(* PLC project MotionTest1, Higen MCL 1 *)
(* stored: creationDateTime 2012-01-06T15:20:13, modificationDateTime 2013-05-16T00:05:34 *)

FUNCTION_BLOCK wxgetval
  VAR
    getpy : python_gear;
    latch : SR;
  END_VAR
  VAR_INPUT
    name : STRING;
  END_VAR
  VAR_OUTPUT
    val : BOOL;
  END_VAR
  VAR  (* added by the conversion: wires and edge detectors of the diagram *)
    _EQ41_ENO : BOOL;
    _EQ41_OUT : BOOL;
    _EQ3_ENO : BOOL;
    _EQ3_OUT : BOOL;
  END_VAR

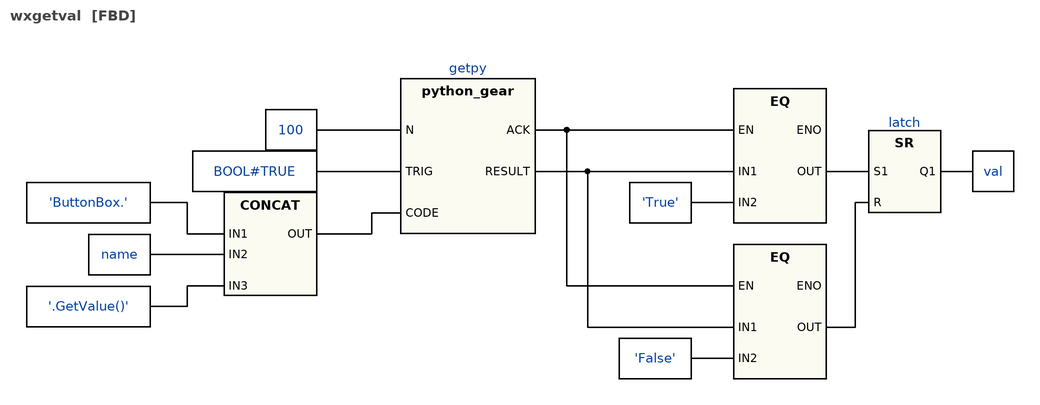
(* FBD diagram, written out as Structured Text *)
getpy(N := 100, TRIG := BOOL#TRUE, CODE := CONCAT('ButtonBox.', name, '.GetValue()'));
_EQ41_OUT := EQ(EN := getpy.ACK, IN1 := getpy.RESULT, IN2 := 'True', ENO => _EQ41_ENO);
_EQ3_OUT := EQ(EN := getpy.ACK, IN1 := getpy.RESULT, IN2 := 'False', ENO => _EQ3_ENO);
latch(S1 := _EQ41_OUT, R := _EQ3_OUT);
val := latch.Q1;
END_FUNCTION_BLOCK

(* -- *)
PROGRAM main
  VAR
    Done : BOOL;
    Slave : AXIS_REF;
    Master1 : AXIS_REF;
    Master2 : AXIS_REF;
    switch : MC_Power;
    readpos : MC_ReadActualPosition;
    sPn : LREAL;
    m1Pn : LREAL;
    m2Pn : LREAL;
    sVn : LREAL;
    m1Vn : LREAL;
    m2Vn : LREAL;
    setpos : MC_SetPosition;
    readspeed : MC_ReadParameter;
    sim : MC_Sim;
    bt1 : wxgetval;
    Block1 : wxgetval;
    Block2 : wxgetval;
    Block3 : wxgetval;
    Block6 : wxgetval;
    MC_Sim0 : MC_Sim;
    MC_Power0 : MC_Power;
    MC_ReadActualPosition0 : MC_ReadActualPosition;
    MC_SetPosition0 : MC_SetPosition;
    MC_ReadParameter0 : MC_ReadParameter;
    MC_MoveAbsolute0 : MC_MoveAbsolute;
    MC_Sim1 : MC_Sim;
    MC_ReadActualPosition1 : MC_ReadActualPosition;
    MC_ReadParameter1 : MC_ReadParameter;
    MC_Power1 : MC_Power;
    MC_SetPosition1 : MC_SetPosition;
    MC_MoveAbsolute1 : MC_MoveAbsolute;
    MC_MoveAbsolute2 : MC_MoveAbsolute;
    MC_MoveAbsolute3 : MC_MoveAbsolute;
    MC_MoveAbsolute4 : MC_MoveAbsolute;
    MC_MoveAbsolute5 : MC_MoveAbsolute;
    MC_CombineAxes0 : MC_CombineAxes;
    MC_Stop0 : MC_Stop;
    MC_Stop1 : MC_Stop;
    MC_Stop2 : MC_Stop;
  END_VAR

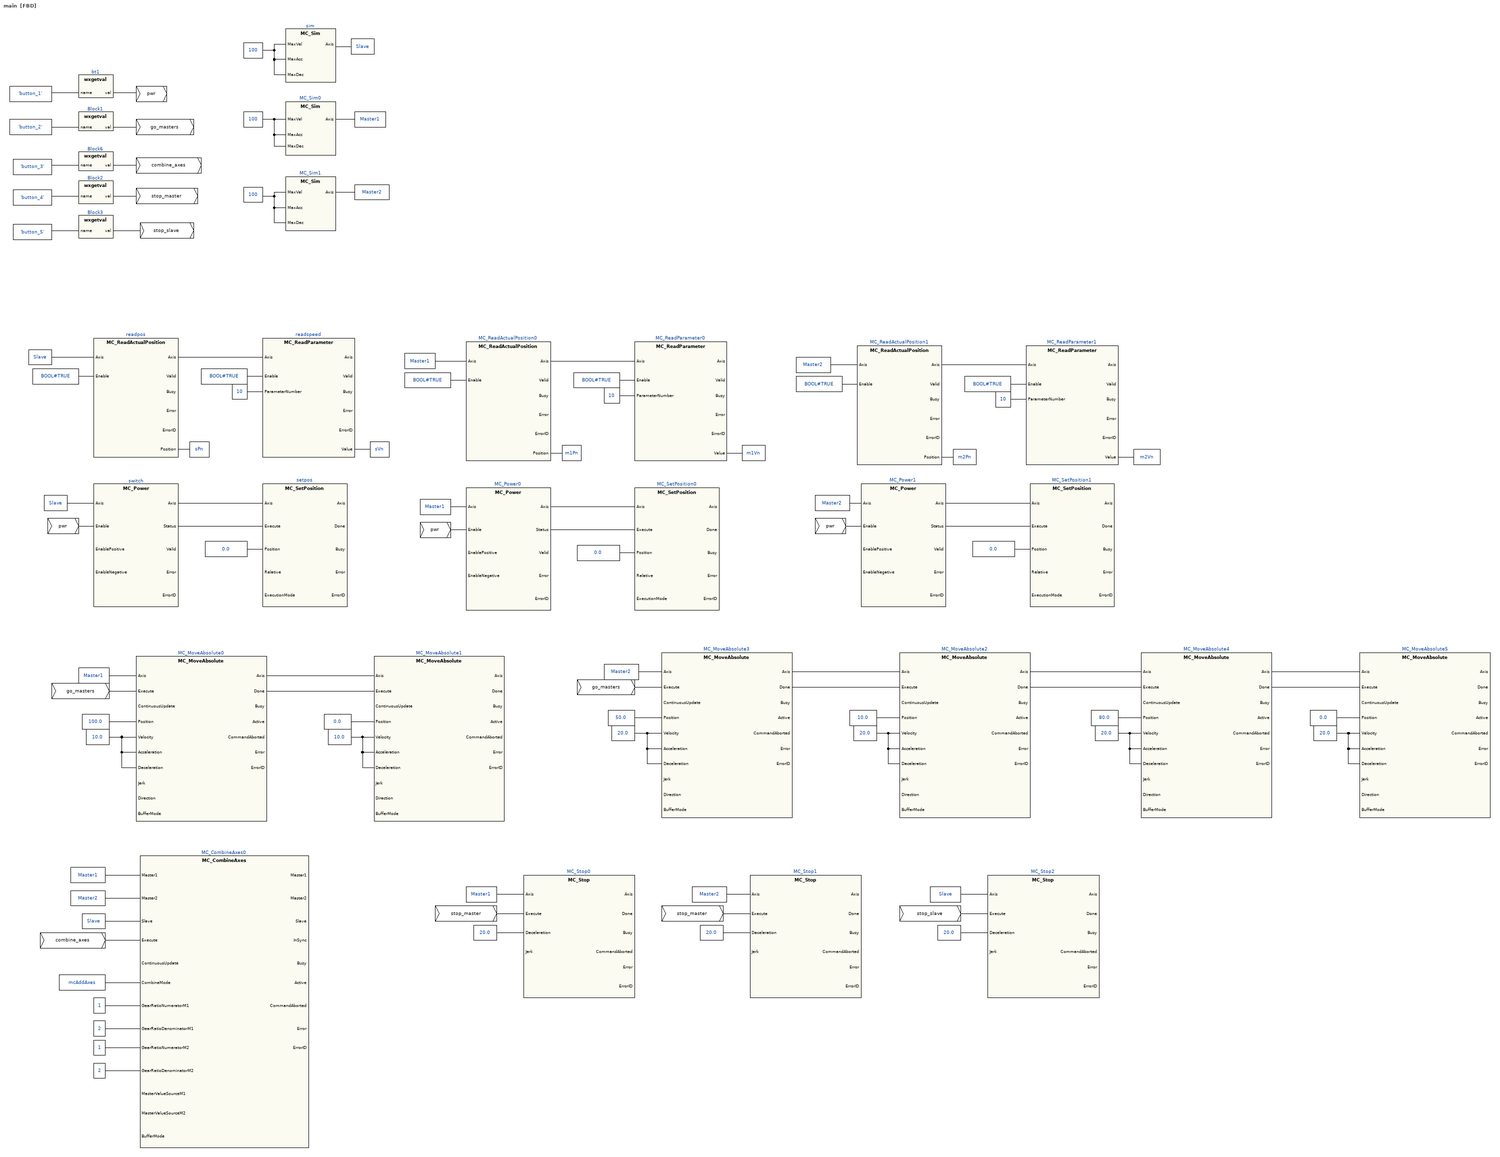
(* FBD diagram, written out as Structured Text *)
sim(MaxVel := 100, MaxAcc := 100, MaxDec := 100);
Slave := sim.Axis;
MC_Sim0(MaxVel := 100, MaxAcc := 100, MaxDec := 100);
Master1 := MC_Sim0.Axis;
MC_Sim1(MaxVel := 100, MaxAcc := 100, MaxDec := 100);
Master2 := MC_Sim1.Axis;
readpos(Axis := Slave, Enable := BOOL#TRUE);
sPn := readpos.Position;
readspeed(Axis := readpos.Axis, Enable := BOOL#TRUE, ParameterNumber := 10);
sVn := readspeed.Value;
MC_ReadActualPosition0(Axis := Master1, Enable := BOOL#TRUE);
m1Pn := MC_ReadActualPosition0.Position;
MC_ReadParameter0(Axis := MC_ReadActualPosition0.Axis, Enable := BOOL#TRUE, ParameterNumber := 10);
m1Vn := MC_ReadParameter0.Value;
MC_ReadActualPosition1(Axis := Master2, Enable := BOOL#TRUE);
m2Pn := MC_ReadActualPosition1.Position;
MC_ReadParameter1(Axis := MC_ReadActualPosition1.Axis, Enable := BOOL#TRUE, ParameterNumber := 10);
m2Vn := MC_ReadParameter1.Value;
bt1(name := 'button_1');
Block1(name := 'button_2');
Block6(name := 'button_3');
Block2(name := 'button_4');
Block3(name := 'button_5');
switch(Axis := Slave, Enable := bt1.val);
setpos(Axis := switch.Axis, Execute := switch.Status, Position := 0.0);
MC_Power0(Axis := Master1, Enable := bt1.val);
MC_SetPosition0(Axis := MC_Power0.Axis, Execute := MC_Power0.Status, Position := 0.0);
MC_Power1(Axis := Master2, Enable := bt1.val);
MC_SetPosition1(Axis := MC_Power1.Axis, Execute := MC_Power1.Status, Position := 0.0);
MC_MoveAbsolute0(Axis := Master1, Execute := Block1.val, Position := 100.0, Velocity := 10.0, Acceleration := 10.0, Deceleration := 10.0);
MC_MoveAbsolute1(Axis := MC_MoveAbsolute0.Axis, Execute := MC_MoveAbsolute0.Done, Position := 0.0, Velocity := 10.0, Acceleration := 10.0, Deceleration := 10.0);
MC_MoveAbsolute3(Axis := Master2, Execute := Block1.val, Position := 50.0, Velocity := 20.0, Acceleration := 20.0, Deceleration := 20.0);
MC_MoveAbsolute2(Axis := MC_MoveAbsolute3.Axis, Execute := MC_MoveAbsolute3.Done, Position := 10.0, Velocity := 20.0, Acceleration := 20.0, Deceleration := 20.0);
MC_MoveAbsolute4(Axis := MC_MoveAbsolute2.Axis, Execute := MC_MoveAbsolute2.Done, Position := 80.0, Velocity := 20.0, Acceleration := 20.0, Deceleration := 20.0);
MC_MoveAbsolute5(Axis := MC_MoveAbsolute4.Axis, Execute := MC_MoveAbsolute4.Done, Position := 0.0, Velocity := 20.0, Acceleration := 20.0, Deceleration := 20.0);
MC_CombineAxes0(Master1 := Master1, Master2 := Master2, Slave := Slave, Execute := Block6.val, CombineMode := mcAddAxes, GearRatioNumeratorM1 := 1, GearRatioDenominatorM1 := 2, GearRatioNumeratorM2 := 1, GearRatioDenominatorM2 := 2);
MC_Stop0(Axis := Master1, Execute := Block2.val, Deceleration := 20.0);
MC_Stop1(Axis := Master2, Execute := Block2.val, Deceleration := 20.0);
MC_Stop2(Axis := Slave, Execute := Block3.val, Deceleration := 20.0);
END_PROGRAM

CONFIGURATION conf
  RESOURCE res ON PLC
    TASK milisecond(INTERVAL := T#10ms, PRIORITY := 0);
    PROGRAM maininstance WITH milisecond : main;
  END_RESOURCE
END_CONFIGURATION
